{attribute addProperty BoxType "EL3773-0000-0018"}
{attribute addProperty Id "I3_SamplesAT %I*ARRAY [1..10] OF INT16020"}
{attribute addProperty CRC "3840097096"}
{attribute addProperty SizeInBites "160"}
{attribute addProperty SizeInBytes "20"}
TYPE L3_Current_Samples_E4E33B48 :
STRUCT
	{attribute addProperty Name "I3_Samples"}
	I3_Samples AT %I* : ARRAY [1..10] OF INT;
END_STRUCT
END_TYPE

(* stored: Version 1.2.0.0, ProductVersion 3.1.4024.9
   DUT L3_Current_Samples_E4E33B48: Id {47be488f-fabc-471d-9286-faf205614de2} *)
